# EPICS substitutions: PIP-II/RFPI2/rfpi-fdr-sw-mgmt-ioc-main/ina-managementApp/Db/slot.substitutions
file board.template {
pattern{ acc, sys, group, num }
{ PIP2IT, pHB650, RFPI, TOP0 }
{ PIP2IT, pHB650, RFPI, TOP1 }
{ PIP2IT, pHB650, RFPI, TOP2 }
{ PIP2IT, pHB650, RFPI, BOT0 }
{ PIP2IT, pHB650, RFPI, BOT1 }
{ PIP2IT, pHB650, RFPI, BOT2 }
{ PIP2IT, pHB650, RFPI, INTER }
{ PIP2IT, pHB650, RFPI, MAIN }
}
